// TIA Portal V19 export
FUNCTION "CoilHandlingMatCounter_CALL" : Void   // FC141, LAD
TITLE = COIL HANDLING MATERIAL COUNTER
// stored: SetENOAutomatically false
   VAR_TEMP
      Stratightener_Standstill : Bool;
   END_VAR
BEGIN

REGION Network 1: Coordination IN
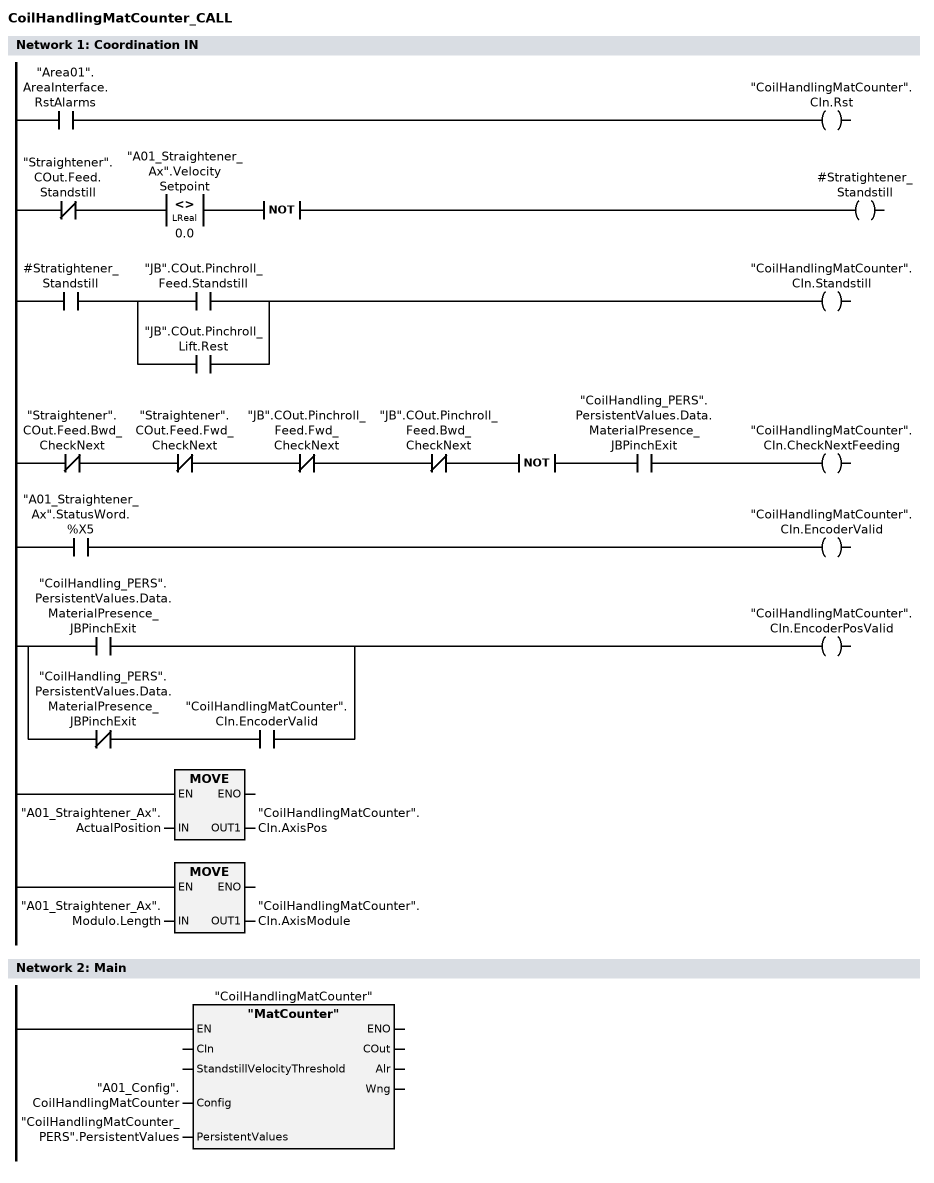
   RUNG wire#powerrail
      Contact( "Area01".AreaInterface.RstAlarms )
      Coil( "CoilHandlingMatCounter".CIn.Rst )
   END_RUNG
   RUNG wire#powerrail
      I_Contact( "Straightener".COut.Feed.Standstill )
      { S7_Templates := "SrcType := LReal" } NE_Contact(in1 := "A01_Straightener_Ax".VelocitySetpoint, in2 := 0.0)
      Not()
      Coil( #Stratightener_Standstill )
   END_RUNG
   RUNG wire#powerrail
      Contact( #Stratightener_Standstill )
      wire#w1
      Contact( "JB".COut.Pinchroll_Feed.Standstill )
      wire#w2
      Coil( "CoilHandlingMatCounter".CIn.Standstill )
   END_RUNG
   RUNG wire#w1
      Contact( "JB".COut.Pinchroll_Lift.Rest )
   END_RUNG wire#w2
   RUNG wire#powerrail
      I_Contact( "Straightener".COut.Feed.Bwd_CheckNext )
      I_Contact( "Straightener".COut.Feed.Fwd_CheckNext )
      I_Contact( "JB".COut.Pinchroll_Feed.Fwd_CheckNext )
      I_Contact( "JB".COut.Pinchroll_Feed.Bwd_CheckNext )
      Not()
      Contact( "CoilHandling_PERS".PersistentValues.Data.MaterialPresence_JBPinchExit )
      Coil( "CoilHandlingMatCounter".CIn.CheckNextFeeding )
   END_RUNG
   RUNG wire#powerrail
      Contact( "A01_Straightener_Ax".StatusWord.%X5 )
      Coil( "CoilHandlingMatCounter".CIn.EncoderValid )
   END_RUNG
   RUNG wire#powerrail
      Contact( "CoilHandling_PERS".PersistentValues.Data.MaterialPresence_JBPinchExit )
      wire#w3
      Coil( "CoilHandlingMatCounter".CIn.EncoderPosValid )
   END_RUNG
   RUNG wire#powerrail
      I_Contact( "CoilHandling_PERS".PersistentValues.Data.MaterialPresence_JBPinchExit )
      Contact( "CoilHandlingMatCounter".CIn.EncoderValid )
   END_RUNG wire#w3
   RUNG wire#powerrail
      { S7_GenerateENO := "TRUE" } Move(in := "A01_Straightener_Ax".ActualPosition, out1 => "CoilHandlingMatCounter".CIn.AxisPos)
   END_RUNG
   RUNG wire#powerrail
      Move(in := "A01_Straightener_Ax".Modulo.Length, out1 => "CoilHandlingMatCounter".CIn.AxisModule)
   END_RUNG
   // the same network as SCL:
   "CoilHandlingMatCounter".CIn.Rst := "Area01".AreaInterface.RstAlarms;
   #Stratightener_Standstill := NOT (NOT "Straightener".COut.Feed.Standstill AND ("A01_Straightener_Ax".VelocitySetpoint <> 0.0));
   "CoilHandlingMatCounter".CIn.Standstill := #Stratightener_Standstill AND ("JB".COut.Pinchroll_Feed.Standstill OR "JB".COut.Pinchroll_Lift.Rest);
   "CoilHandlingMatCounter".CIn.CheckNextFeeding := NOT (NOT "Straightener".COut.Feed.Bwd_CheckNext AND NOT "Straightener".COut.Feed.Fwd_CheckNext AND NOT "JB".COut.Pinchroll_Feed.Fwd_CheckNext AND NOT "JB".COut.Pinchroll_Feed.Bwd_CheckNext) AND "CoilHandling_PERS".PersistentValues.Data.MaterialPresence_JBPinchExit;
   "CoilHandlingMatCounter".CIn.EncoderValid := "A01_Straightener_Ax".StatusWord.%X5;
   "CoilHandlingMatCounter".CIn.EncoderPosValid := "CoilHandling_PERS".PersistentValues.Data.MaterialPresence_JBPinchExit OR (NOT "CoilHandling_PERS".PersistentValues.Data.MaterialPresence_JBPinchExit AND "CoilHandlingMatCounter".CIn.EncoderValid);
   "CoilHandlingMatCounter".CIn.AxisPos := "A01_Straightener_Ax".ActualPosition;
   "CoilHandlingMatCounter".CIn.AxisModule := "A01_Straightener_Ax".Modulo.Length;
END_REGION

REGION Network 2: Main
   RUNG wire#powerrail
      "CoilHandlingMatCounter"(CIn :=, StandstillVelocityThreshold :=, Config := "A01_Config".CoilHandlingMatCounter, PersistentValues := "CoilHandlingMatCounter_PERS".PersistentValues, COut =>, Alr =>, Wng =>)
   END_RUNG
   // the same network as SCL:
   "CoilHandlingMatCounter"(Config := "A01_Config".CoilHandlingMatCounter,   // "MatCounter"
                           PersistentValues := "CoilHandlingMatCounter_PERS".PersistentValues);
END_REGION

REGION Network 3: >
END_REGION

REGION Network 4: >
END_REGION

REGION Network 5: >
END_REGION
END_FUNCTION
